INTERFACE I_WorkingStation

METHOD mErrorReset : BOOL
VAR_INPUT
END_VAR
END_METHOD

PROPERTY prEmptyMode : BOOL
GET
END_GET
SET
END_SET
END_PROPERTY

PROPERTY prError : BOOL
GET
END_GET
END_PROPERTY

PROPERTY prErrorNumber : UDINT
GET
END_GET
END_PROPERTY

PROPERTY prInManualMode : BOOL
GET
END_GET
END_PROPERTY

PROPERTY prIsEmpty : BOOL
GET
END_GET
END_PROPERTY

PROPERTY prTablePlace : REFERENCE TO FB_TablePlace
GET
END_GET
SET
END_SET
END_PROPERTY

{attribute 'monitoring' := 'call'}
PROPERTY prTableRotationInterlock : BOOL
GET
END_GET
SET
END_SET
END_PROPERTY

{attribute 'monitoring' := 'call'}
PROPERTY prTableRotationRequest : BOOL
GET
END_GET
END_PROPERTY

END_INTERFACE

(* stored: Version 1.1.0.1, ProductVersion 3.1.4024.15
   Itf I_WorkingStation: Id {4fc3fe90-c1e8-40cd-ba9f-deea71f0ae85}
   Method mErrorReset: Id {f1df3791-fffd-46bd-a138-b8731344e2cf}
   Property prEmptyMode: Id {61a49ff7-8236-4462-8d7c-d1dd0f63e4ad}
   Get Get: Id {affb2f8a-5102-4174-a6db-da1bf06d7008}
   Set Set: Id {a201dae3-9df4-4ef9-a161-aca13abce986}
   Property prError: Id {341f54d4-cb33-4e29-9291-db8b8afe04b9}
   Get Get: Id {dbc2c9cd-1825-4cc1-850f-d37b416451ca}
   Property prErrorNumber: Id {3ad9980e-dc87-4b73-aca5-009facae308e}
   Get Get: Id {d2af7160-dedf-446b-8cc9-0b9c6dee0edc}
   Property prInManualMode: Id {364ecbd4-c120-41ba-8855-bf61cc714345}
   Get Get: Id {7c028eb7-8db4-402e-9f37-9908d59bc3de}
   Property prIsEmpty: Id {48a9aebc-d01f-4528-9b85-4b769b9e0034}
   Get Get: Id {e161129c-8418-48d3-81fe-587141a41b59}
   Property prTablePlace: Id {dfd52d25-5a09-44cb-bdb3-a50f7756e0ee}
   Get Get: Id {3d238b09-2f8f-44c4-9ef4-69991e9b0500}
   Set Set: Id {57812a8e-8d13-421a-bfd6-20c58ef44f42}
   Property prTableRotationInterlock: Id {36e7e1ef-3eca-4e02-9d42-157e2e1fc858}
   Get Get: Id {01bd09b6-9f54-4c2d-b79d-742c5fdb82f3}
   Set Set: Id {dd8d538d-614e-475f-a33a-115fd16c76f1}
   Property prTableRotationRequest: Id {ad483de5-b236-4c2c-82fd-5d0976a0b1c1}
   Get Get: Id {add0ad2f-100e-4e6f-9dce-4eb57c7d81e1} *)
